// TIA Portal V16 export
// export: Created 2021-03-04T22:04:04.6024191Z, ExportSetting WithDefaults, DisplayName Totally Integrated Automation Portal, DisplayVersion V16, DisplayName TIA Portal Version Control Interface, DisplayVersion V16, DisplayName TIA Portal Openness, DisplayVersion V16, DisplayName SINAMICS Startdrive Advanced, DisplayVersion V16, DisplayName SINAMICS Startdrive G130, G150, S120, S150, SINAMICS MV, S210, DisplayVersion V16, DisplayName SINAMICS Startdrive G110M, G120, G120C, G120D, G120P, DisplayVersion V16, DisplayName STEP 7 Professional, DisplayVersion V16, DisplayName STEP 7 Safety, DisplayVersion V16, DisplayName WinCC Professional, DisplayVersion V16
VAR_GLOBAL   // PLC tag table "IO"
   GlobalAI AT %I100.0 : "udtArrAIGlobal";   //    {ExternalAccessible false, ExternalVisible false, ExternalWritable false}
   GlobalDQ AT %Q100.0 : "udtArrDQGlobal";   //    {ExternalAccessible false, ExternalVisible false, ExternalWritable false}
END_VAR
